Universal Robots PolyScope program: nastro 30 maggio.urp

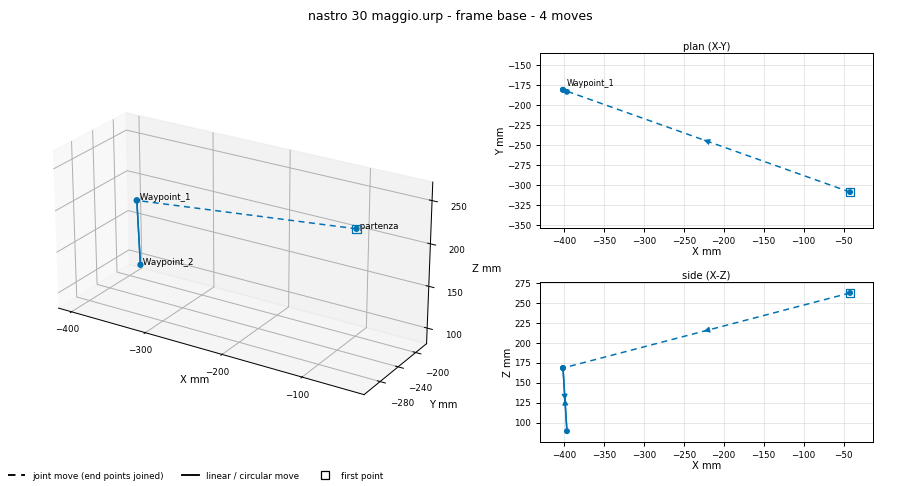
[picture p0: tool path of nastro 30 maggio.urp in frame base, 4 of 4 moves have a stored position in this frame; points joined in program order, loops and branches not executed]
Program nastro 30 maggio (installation=default directory=/programs createdIn=3.15.3.106223 lastSavedIn=3.15.8.106339 robotSerialNumber=2021330429)
Calibrated DH parameters: a=[-0.000156, -0.236402, -0.171625, 0.000006, -0.000047, 0]; d=[0.151683, 29.702709, 78.973085, -108.563557, 0.085229, 0.082167]; alpha=[1.57015, 0.001987, 0.001164, 1.571718, -1.571778, 0]; deltaTheta=[-0.000066, 0.24449, 0.39032, -0.635025, 0.000068, -0.000043]
BeforeStart
  cont := 0
  URCap Gripper Activate (Robotiq_Grippers, Robotiq Inc.) dataModel(ResetAndActivateKey=false)
  ready := False
  Timer (action=Stop) variable(name=volo)
  URCap Gripper (Robotiq_Grippers, Robotiq Inc.) dataModel(position=34.509803921568626, force=0.0, speed=0.0, positionInDouble=34.509803921568626, forceInDouble=0.0, speedInDouble=0.0, slaveIds=[9], blocking=true)
Robot Program (runOnlyOnce=false)
  Wait Condition expression=ready≟ True
  MoveJ speed 60 deg/s, acceleration 80 deg/s^2 (useActiveTCP=true)
    Waypoint partenza: TCP in base x=-41.997 y=-308.663 z=263.002 mm, rx=0.0045 ry=3.0917 rz=0.0492 rad; joints [280.902, -97.845, -50.961, -122.382, 93.173, 370.919] deg; flange x=-49.773 y=-313.645 z=419.733 mm, rx=0.0047 ry=3.0917 rz=0.0492 rad
    Waypoint Waypoint_1: TCP in base x=-401.064 y=-180.745 z=168.671 mm, rx=-0.035 ry=3.1297 rz=0.0792 rad; joints [220.139, -126.323, -36.573, -109.35, 88.266, 308.781] deg; flange x=-402.662 y=-188.7 z=325.462 mm, rx=-0.035 ry=3.1297 rz=0.0792 rad
  MoveL speed 250 mm/s, acceleration 1200 mm/s^2 (useActiveTCP=true) feature=Base
    Waypoint Waypoint_2: TCP in base x=-396.098 y=-183.244 z=89.293 mm, rx=-0.0351 ry=3.1297 rz=0.0791 rad; joints [220.835, -123.021, -63.621, -85.626, 88.307, 309.49] deg; flange x=-397.693 y=-191.197 z=246.084 mm, rx=-0.0351 ry=3.1297 rz=0.0791 rad
    URCap Gripper (Robotiq_Grippers, Robotiq Inc.) dataModel(position=100.0, force=0.0, speed=0.0, positionInDouble=100.0, forceInDouble=0.0, speedInDouble=0.0, slaveIds=[9], blocking=true)
    Waypoint Waypoint_3: TCP in base x=-401.063 y=-180.748 z=168.669 mm, rx=-0.035 ry=3.1296 rz=0.0791 rad; joints [220.139, -126.324, -36.573, -109.35, 88.268, 308.781] deg; flange x=-402.664 y=-188.699 z=325.46 mm, rx=-0.035 ry=3.1296 rz=0.0791 rad
  Pallet pattern(dimensionality=Box firstAxisCount=2 secondAxisCount=2 thirdAxisCount=2 motionType=MoveL speed=0.25 acceleration=1.2 useActiveTCP=true, counterVariable(name=cnt_1, initializeExpression=0), patternPoseVariable(name=pose_1), feature=Base, children(Waypoint(type=Fixed name=Corner1_1, position(joints=5.072078227996826, -2.1095407644854944, -1.6215422789203089, -0.9462693373309534, 1.6097885370254517, 6.7470279971705835 pose=0.04170376535466645, -0.4064286791616084, 0.006640908341733531, 0.16155953542922305, 3.0901611511753737, -0.025331480643686517), poseInFeatureCoordinates=[0.041704, -0.406429, 0.006641, 0.16156, 3.090161, -0.025331], outputFlangePose=[0.034455, -0.403477, 0.163446, 0.16156, 3.090161, -0.025331]), Waypoint(type=Fixed name=Corner2_1, position(joints=4.956535339355469, -2.069923226033346, -1.6320775190936487, -1.000817600880758, 1.5708147287368774, 6.574159298335211 pose=-0.017118488693580538, -0.40004045105256786, 0.014162335191012954, 0.07527521301985846, 3.1406032927752006, -0.01361095451125088), poseInFeatureCoordinates=[-0.017118, -0.40004, 0.014162, 0.075275, 3.140603, -0.013611], outputFlangePose=[-0.017095, -0.39868, 0.171156, 0.075275, 3.140603, -0.013611]), Waypoint(type=Fixed name=Corner3_1, position(joints=5.1470842361450195, -1.9763882795916956, -1.7892840544330042, -0.9720137755023401, 1.5684523582458496, 6.778223309909002 pose=0.043180393955634326, -0.3632071880339587, 0.009949401333471108, -0.095968893820628, -3.1241534150248844, -0.03395845698980473), poseInFeatureCoordinates=[0.04318, -0.363207, 0.009949, -0.095969, -3.124153, -0.033958], outputFlangePose=[0.045552, -0.366692, 0.166893, -0.095969, -3.124153, -0.033958]), Waypoint(type=Fixed name=Corner4_1, position(joints=5.027559757232666, -1.9602497259723108, -1.8051188627826136, -0.9944742361651819, 1.5497816801071167, 6.699367497359411 pose=-0.0074393736274557505, -0.3586289829127899, 0.009893055179691551, -0.15760636692063246, -3.0982006147387295, -0.057766086249757535), poseInFeatureCoordinates=[-0.007439, -0.358629, 0.009893, -0.157606, -3.098201, -0.057766], outputFlangePose=[-0.001648, -0.364774, 0.166666, -0.157606, -3.098201, -0.057766]), Waypoint(type=Fixed name=Corner5_1, position(joints=5.072066307067871, -2.043708626423971, -1.5555079619037073, -1.0781033674823206, 1.6095963716506958, 6.746859852467672 pose=0.04168701531055582, -0.4064429099486951, 0.03872495077040053, 0.1616155807489969, 3.0901922020862727, -0.025421877378065946), poseInFeatureCoordinates=[0.041687, -0.406443, 0.038725, 0.161616, 3.090192, -0.025422], outputFlangePose=[0.034444, -0.403483, 0.19553, 0.161616, 3.090192, -0.025422]), Waypoint(type=Fixed name=Corner6_1, position(joints=4.95648717880249, -2.0162022749530237, -1.5723555723773401, -1.11424428621401, 1.570658564567566, 6.573991511260168 pose=-0.0171483620840403, -0.4000438888775143, 0.0412719046186856, 0.07533336053907952, 3.1406327482211815, -0.013650511432852154), poseInFeatureCoordinates=[-0.017148, -0.400044, 0.041272, 0.075333, 3.140633, -0.013651], outputFlangePose=[-0.01712, -0.39868, 0.198266, 0.075333, 3.140633, -0.013651]), Waypoint(type=Fixed name=Corner7_1, position(joints=5.147120475769043, -1.9091947714435022, -1.7207329908954065, -1.107899014149801, 1.568296194076538, 6.7780791262732905 pose=0.043172541157023396, -0.3631804323712314, 0.04042768630534191, -0.09595109257338075, -3.1240819741556107, -0.0341495504154411), poseInFeatureCoordinates=[0.043173, -0.36318, 0.040428, -0.095951, -3.124082, -0.03415], outputFlangePose=[0.045554, -0.366685, 0.19737, -0.095951, -3.124082, -0.03415]), Waypoint(type=Fixed name=Corner8_1, position(joints=5.027631759643555, -1.8940032164203089, -1.7368577162372034, -1.1288912932025355, 1.54954195022583, 6.699235651885168 pose=-0.0074349826122077824, -0.3586548243383853, 0.03984157990237988, -0.15753958584666863, -3.098153545436267, -0.057586709775178), poseInFeatureCoordinates=[-0.007435, -0.358655, 0.039842, -0.15754, -3.098154, -0.057587], outputFlangePose=[-0.001634, -0.364782, 0.196615, -0.15754, -3.098154, -0.057587]))); actionSequence(name=PalletSequence motionType=MoveL speed=0.25 acceleration=1.2 useActiveTCP=true, anchorWaypoint(type=Fixed name=PatternPoint_1, position(joints=5.07218599319458, -2.065842930470602, -1.5818122068988245, -1.0296242872821253, 1.6097406148910522, 6.746895794068472 pose=0.04175901220671263, -0.40643278798117577, 0.027076785175474904, 0.16137201437998652, 3.09010176666312, -0.025412789297814126), poseInFeatureCoordinates=[0.041759, -0.406433, 0.027077, 0.161372, 3.090102, -0.025413], outputFlangePose=[0.0345, -0.403473, 0.183881, 0.161372, 3.090102, -0.025413]), feature=Base, children(Waypoint(type=Fixed name=Approach_1, position(joints=5.072078227996826, -1.9670088926898401, -1.3908847014056605, -1.3194921652423304, 1.6094286441802979, 6.746523920689718 pose=0.04169836636926619, -0.4064222669655773, 0.0949922155470864, 0.16154768820106188, 3.090168938754823, -0.025312134352228725), poseInFeatureCoordinates=[0.041698, -0.406422, 0.094992, 0.161548, 3.090169, -0.025312], outputFlangePose=[0.034451, -0.403473, 0.251797, 0.161548, 3.090169, -0.025312]), Waypoint=PatternPoint_1, Contributed(strategyProgramNodeType=Gripper strategyURCapDeveloper=Robotiq Inc. strategyURCapName=Robotiq_Grippers, dataModel(position=0.0, force=0.0, speed=0.0, positionInDouble=0.0, forceInDouble=0.0, speedInDouble=0.0, slaveIds=[9], blocking=true)), Wait(type=Sleep, waitTime=1), Waypoint(type=Fixed name=Exit_1, position(joints=5.072054386138916, -1.967104736958639, -1.390836540852682, -1.319552246724264, 1.609344720840454, 6.7465718428241175 pose=0.04166775688550932, -0.40642465525955396, 0.0949625080191086, 0.1616704481804114, 3.090283335420461, -0.025211262699491203), poseInFeatureCoordinates=[0.041668, -0.406425, 0.094963, 0.16167, 3.090283, -0.025211], outputFlangePose=[0.034438, -0.403486, 0.251768, 0.16167, 3.090283, -0.025211])))
    Pattern -> pattern
    AnchoredSequence -> PalletSequence
Thread Thread_1 (runOnlyOnce=false)
  If digital_in[4]
    Set DigitalOutput pin=digital_out[0]; digitalValue=1
    Timer (action=Start) variable=volo
    Timer (action=Reset) variable=volo
    Wait DigitalInput pin=digital_in[4]; digitalValue=0
  ElseIf digital_in[5]
    Wait Sleep waitTime=0.3
    Set DigitalOutput pin=digital_out[0]; digitalValue=0
    ready := True
    Wait DigitalInput pin=digital_in[5]; digitalValue=0
    Set DigitalOutput pin=digital_out[0]; digitalValue=1
    ready := False
    Timer (action=Start) variable=volo
    Timer (action=Reset) variable=volo
  If volo>10
    Timer (action=Stop) variable=volo
    Timer (action=Reset) variable=volo
    Set DigitalOutput pin=digital_out[0]; digitalValue=0
